{attribute 'GeneratedUsingTerminal: EJ7211-0011-0026'}
{attribute addProperty BoxType "EJ7211-0011-0026"}
{attribute addProperty Id "StatuswordAT %I*UINT2"}
{attribute addProperty CRC "2604072444"}
{attribute addProperty Size "2"}
TYPE DS402_Statusword_9B36FDFC EXTENDS InputBase_8311D824 :
STRUCT
	{attribute addProperty Name "Statusword"}
	Statusword AT %I* : UINT;
END_STRUCT
END_TYPE

(* stored: Version 1.2.0.0, ProductVersion 3.1.4024.9
   DUT DS402_Statusword_9B36FDFC: Id {999074eb-4060-4c4d-be82-abbff576ec3e} *)
